// TIA Portal project "pickAndPlace" (V15)
// Ejemplo didactico

(* hardware
DEVICE "HMI_1"  TP700 Comfort
   slot 0: "HMI_1"  TP700 Comfort  6AV2 124-0GC01-0AX0  15.0.0.0
   slot 1: "HMI_RT_1"  TP700 Comfort  6AV2 124-0GC01-0AX0  15.0.0.0
   slot 5: "HMI_1.IE_CP_1"  PROFINET Interface  15.0.0.0
      slot 1: "Interfaz PROFINET_1"  PROFINET Interface
         slot 1: "Port_1"  Port
         slot 2: "Port_2"  Port
   slot 7: "HMI_1.MPI/DP_CP_1"  MPI/DP Interface  15.0.0.0
DEVICE "S7-1200 station_1"  S7-1200 Station
   slot 0: "Rack_0"  S7-1200 Rack  Rack  V1.0
   slot 1: "PLC_1"  CPU 1214C AC/DC/Rly  6ES7 214-1BG40-0XB0  V4.2
*)

// ===== PLC "PLC_1"  CPU 1214C AC/DC/Rly =====

VAR_GLOBAL   // PLC tag table "Tabla de variables estándar"
   "inicio" AT %M0.0 : Bool;
   "motor1" AT %Q0.1 : Bool;
   "animacionBotella" AT %MW2 : Int;
   "resetTimeBotella" AT %M0.1 : Bool;
   "paso2" AT %M0.2 : Bool;
   "setBotellasEnCaja" AT %MW4 : Int;
   "paso1" AT %M0.3 : Bool;
   "resetContadorBotellas" AT %M0.4 : Bool;
   "botellasActualesEnCaja" AT %MW6 : Int;
   "triggerInicio" AT %M0.5 : Bool;
   "animacionElevador" AT %MW8 : Int;
   "resetTimeElevador" AT %M0.6 : Bool;
   "paso3" AT %M0.7 : Bool;
   "animacionCaja" AT %MW10 : Int;
   "resetTimeCaja" AT %M1.0 : Bool;
   "fin" AT %M1.1 : Bool;
   "preFin" AT %M1.2 : Bool;
END_VAR

// folder: System blocks/Program resources

DATA_BLOCK "timeBotella"   // DB1
{ S7_Optimized_Access := 'TRUE' }
AUTHOR : Simatic
FAMILY : IEC
NAME : IEC_TMR
VERSION : 1.0
// stored: InstanceOfName IEC_TIMER
"IEC_TIMER"
BEGIN
END_DATA_BLOCK

DATA_BLOCK "botellasEnCaja"   // DB2
{ S7_Optimized_Access := 'TRUE' }
AUTHOR : Simatic
FAMILY : IEC
NAME : CNTR
VERSION : 1.0
// stored: InstanceOfName IEC_COUNTER
"IEC_COUNTER"
BEGIN
END_DATA_BLOCK

DATA_BLOCK "timeElevador"   // DB3
{ S7_Optimized_Access := 'TRUE' }
AUTHOR : Simatic
FAMILY : IEC
NAME : IEC_TMR
VERSION : 1.0
// stored: InstanceOfName IEC_TIMER
"IEC_TIMER"
BEGIN
END_DATA_BLOCK

DATA_BLOCK "timeCaja"   // DB4
{ S7_Optimized_Access := 'TRUE' }
AUTHOR : Simatic
FAMILY : IEC
NAME : IEC_TMR
VERSION : 1.0
// stored: InstanceOfName IEC_TIMER
"IEC_TIMER"
BEGIN
END_DATA_BLOCK

DATA_BLOCK "timeFin"   // DB5
{ S7_Optimized_Access := 'TRUE' }
AUTHOR : Simatic
FAMILY : IEC
NAME : IEC_TMR
VERSION : 1.0
// stored: InstanceOfName IEC_TIMER
"IEC_TIMER"
BEGIN
END_DATA_BLOCK

// folder: (top level)

ORGANIZATION_BLOCK "Main"   // OB1, LAD, ProgramCycle
TITLE = "Main Program Sweep (Cycle)"
{ S7_Optimized_Access := 'TRUE' }
VERSION : 0.1
   VAR_INPUT
      Initial_Call : Bool;   // Initial call of this OB
      Remanence : Bool;   // =True, if remanent data are available
   END_VAR
   VAR_TEMP   // added for the SCL form of the ladder/FBD networks
      _w1 : Bool;
      _w2 : Bool;
      _w3 : Bool;
   END_VAR
BEGIN

REGION Network 2: Condiciones iniciales
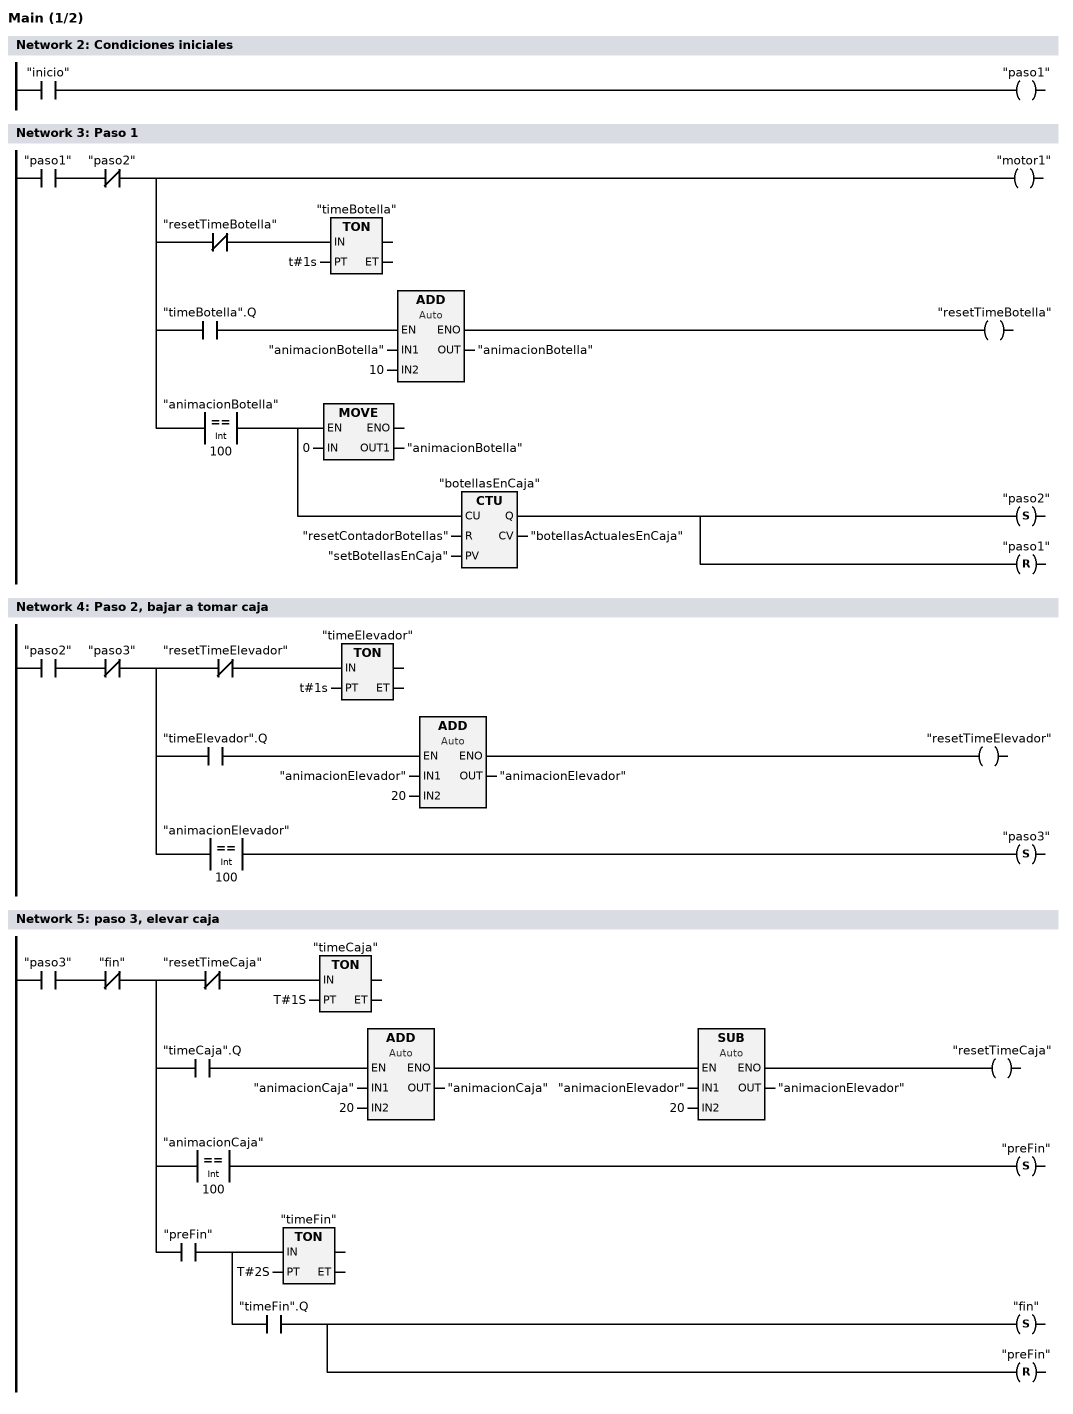
   RUNG wire#powerrail
      Contact( "inicio" )
      Coil( "paso1" )
   END_RUNG
   // the same network as SCL:
   "paso1" := "inicio";
END_REGION

REGION Network 3: Paso 1
   "motor1" := "paso1" AND NOT "paso2";
   "timeBotella".TON(IN := "motor1" AND NOT "resetTimeBotella", PT := t#1s);
   #_w1 := "motor1" AND "timeBotella".Q;
   IF #_w1 THEN "animacionBotella" := "animacionBotella" + 10; END_IF;
   "resetTimeBotella" := #_w1;
   #_w2 := "motor1" AND ("animacionBotella" = 100);
   IF #_w2 THEN "animacionBotella" := 0; END_IF;
   "botellasEnCaja".CTU(CU := #_w2,
                        R := "resetContadorBotellas",
                        PV := "setBotellasEnCaja",
                        CV => "botellasActualesEnCaja");
   IF "botellasEnCaja".Q THEN
       "paso2" := TRUE;
       "paso1" := FALSE;
   END_IF;
END_REGION

REGION Network 4: Paso 2, bajar a tomar caja
   #_w1 := "paso2" AND NOT "paso3";
   "timeElevador".TON(IN := #_w1 AND NOT "resetTimeElevador", PT := t#1s);
   #_w2 := #_w1 AND "timeElevador".Q;
   IF #_w2 THEN "animacionElevador" := "animacionElevador" + 20; END_IF;
   "resetTimeElevador" := #_w2;
   IF #_w1 AND ("animacionElevador" = 100) THEN "paso3" := TRUE; END_IF;
END_REGION

REGION Network 5: paso 3, elevar caja
   #_w1 := "paso3" AND NOT "fin";
   "timeCaja".TON(IN := #_w1 AND NOT "resetTimeCaja", PT := T#1S);
   #_w2 := #_w1 AND "timeCaja".Q;
   IF #_w2 THEN
       "animacionCaja" := "animacionCaja" + 20;
       "animacionElevador" := "animacionElevador" - 20;
   END_IF;
   "resetTimeCaja" := #_w2;
   IF #_w1 AND ("animacionCaja" = 100) THEN "preFin" := TRUE; END_IF;
   #_w3 := #_w1 AND "preFin";
   "timeFin".TON(IN := #_w3, PT := T#2S);
   IF #_w3 AND "timeFin".Q THEN
       "fin" := TRUE;
       "preFin" := FALSE;
   END_IF;
END_REGION

REGION Network 6: fin
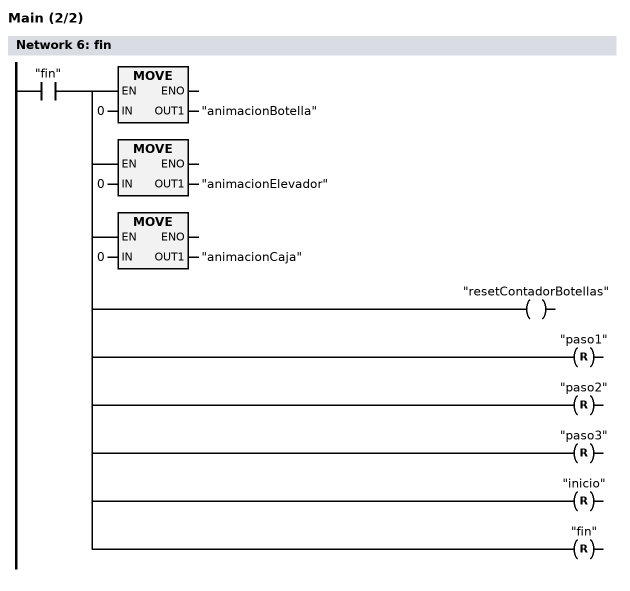
   RUNG wire#powerrail
      Contact( "fin" )
      wire#w1
      Move(in := 0, out1 => "animacionBotella")
   END_RUNG
   RUNG wire#w1
      Move(in := 0, out1 => "animacionElevador")
   END_RUNG
   RUNG wire#w1
      Move(in := 0, out1 => "animacionCaja")
   END_RUNG
   RUNG wire#w1
      Coil( "resetContadorBotellas" )
   END_RUNG
   RUNG wire#w1
      R_Coil( "paso1" )
   END_RUNG
   RUNG wire#w1
      R_Coil( "paso2" )
   END_RUNG
   RUNG wire#w1
      R_Coil( "paso3" )
   END_RUNG
   RUNG wire#w1
      R_Coil( "inicio" )
   END_RUNG
   RUNG wire#w1
      R_Coil( "fin" )
   END_RUNG
   // the same network as SCL:
   IF "fin" THEN
       "animacionBotella" := 0;
       "animacionElevador" := 0;
       "animacionCaja" := 0;
   END_IF;
   "resetContadorBotellas" := "fin";
   IF "fin" THEN
       "paso1" := FALSE;
       "paso2" := FALSE;
       "paso3" := FALSE;
       "inicio" := FALSE;
       "fin" := FALSE;
   END_IF;
END_REGION
END_ORGANIZATION_BLOCK

(* ===== HMI "HMI_RT_1" =====
system functions are stored by id; their names below are inferred from use
connection "HMI_Conexión_1": ETHERNET, S7_1200_OMS

HMI tags "Tabla de variables estándar"
   "Número_imagen_variable" : UInt, internal
   "inicio" : Bool = PLC inicio AT %M0.0, 1 s
   "motor1" : Bool = PLC motor1 AT %Q0.1, 1 s
   "animacionBotella" : Int = PLC animacionBotella AT %MW2, 1 s
   "setBotellasEnCaja" : Int = PLC setBotellasEnCaja AT %MW4, 1 s
   "botellasActualesEnCaja" : Int = PLC botellasActualesEnCaja AT %MW6, 1 s
   "animacionElevador" : Int = PLC animacionElevador AT %MW8, 1 s
   "animacionCaja" : Int = PLC animacionCaja AT %MW10, 1 s

text list "Nombre_imagen_lista_texto": 1 'Imagen raíz'

screen "Imagen raíz" 800x420, template "Plantilla_1"
   on GenerateScreen: SetTag("Número_imagen_variable", 1)
   GraphicView "Visor de gráficos_1" at 30,311 size 54x48; Picture "Gráfico_1"
   GraphicView "Visor de gráficos_4" at 70,300 size 534x53; Picture "Gráfico_7"
   GraphicView "Visor de gráficos_5" at 585,3 size 138x148; Picture "Gráfico_12"
      VerticalMovement <- "animacionElevador"
   GraphicView "Visor de gráficos_2" at 132,261 size 19x63; Picture "Gráfico_13"
      HorizontalMovement <- "animacionBotella"
   GraphicView "Visor de gráficos_3" at 599,235 size 108x82; Picture "Gráfico_14"
      VerticalMovement <- "animacionCaja"
   GraphicView "Visor de gráficos_6" at 585,311 size 118x59; Picture "Gráfico_18"
   TextField "Campo de texto_1" at 29,287 size 38x23; Text 'OFF'
      Visibility <- "motor1"
   TextField "Campo de texto_2" at 32,287 size 31x23; Text 'ON'
      Visibility <- "motor1"
   Button "Botón_1" at 13,42 size 96x32; TextOff 'START'
      on Click: SetBit("inicio")
      Visibility <- "inicio"
   Button "Botón_2" at 13,41 size 96x32; TextOff 'STOP'
      on Click: ResetBit("inicio")
      Visibility <- "inicio"
   TextField "Campo de texto_3" at 8,3 size 204x23; Text 'Simple Pick and Place'
   Circle "Círculo_1" at 129,42 size 34x34
      Appearance <- "inicio"
   TextField "Campo de texto_4" at 20,127 size 175x23; Text 'Botellas por Caja:'
   IOField "Campo ES_1" at 201,123 size 44x32; FormatPattern 99
      ProcessValue <- "setBotellasEnCaja"
   IOField "Campo ES_2" at 723,269 size 41x32; FormatPattern 99
      ProcessValue <- "botellasActualesEnCaja"

Template "Plantilla_1" 800x420
   Button "Salir" at 720,385 size 78x33; TextOff 'Salir'; PictureOff "ExitRuntime_TP700_Comfort_TR"; PictureOn "ExitRuntime_TP700_Comfort_TR"
      on Release: StopRuntime(0)
   Button "Template_Button" at 640,385 size 78x33; TextOff 'Text'
   Button "Template_Button_1" at 560,385 size 78x33; TextOff 'Text'
   Button "Template_Button_2" at 480,385 size 78x33; TextOff 'Text'
   Button "Template_Button_3" at 400,385 size 78x33; TextOff 'Text'
   Button "Template_Button_4" at 321,385 size 78x33; TextOff 'Text'
   Button "Template_Button_5" at 241,385 size 78x33; TextOff 'Text'
   Button "Template_Button_6" at 161,385 size 78x33; TextOff 'INFO'
      on Click: ActivateScreen("info", 0)
   Button "Avisos" at 81,385 size 78x33; TextOff 'Avisos'; PictureOff "AlarmDisplay_TP700_Comfort_TR"; PictureOn "AlarmDisplay_TP700_Comfort_TR"
      on Release: function_ef3f5d25("Ventana de avisos_no_acusado", -1)
   Button "Imagen inicial" at 1,385 size 78x33; TextOff 'Imagen inicial'; PictureOff "NavigateHome_TP700_Comfort_TR"; PictureOn "NavigateHome_TP700_Comfort_TR"
      on Release: ActivateScreen("Imagen raíz", 0)

screen "info" 800x420, template "Plantilla_1"
   TextField "Campo de texto_1" at 55,24 size 274x29; Text 'Descripcion del sistema'
   TextField "Campo de texto_2" at 58,77 size 679x23; Text 'Seteos previos: Colocar la cantidad de botellas que deben ir en cada caja.'
   TextField "Campo de texto_3" at 57,104 size 663x61; Text 'Paso 1: Al hacer ckic en START se enciende lampara en Verde indicando sistema en funcionamiento, se energiza el motor M1 y las botellas comienzan a ingresar a la caja hasta alcanzar la cantidad seteada.'
   TextField "Campo de texto_4" at 59,168 size 589x42; Text 'Paso 2:Una vez completa la caja, procede a bajar el brazo para posicionarse y tomar la caja.'
   TextField "Campo de texto_5" at 60,215 size 539x42; Text 'Paso 3:El elevador sube la caja y da final al ciclo al llegar arriba y alli queda esperando por un nuevo inicio.'
*)